FUNCTION_BLOCK AutomaticFB
VAR_INPUT
END_VAR
VAR_OUTPUT
END_VAR
VAR
END_VAR

// NETWORK 1

END_FUNCTION_BLOCK

(* stored: Version 1.1.0.1, ProductVersion 3.1.4024.15
   POU AutomaticFB: Id {eaf3527e-b7cb-4771-b749-2b4a4935e78a}, SpecialFunc None *)
